// TIA Portal V18 export
DATA_BLOCK "FB_MES_Monitoring_iDB"   // DB10
// stored: InstanceOfName FB_MES_Monitoring, InstanceOfType FB
"FB_MES_Monitoring"
   // VAR_INPUT
   //    Enable : Bool;
   //    Reset : Bool;
   //    HeartbeatTimeout_MES : Time;
   //    HeartbeatTimeout_PLC : Time;
   //    CheckInTimeout : Time;
   //    CheckOutTimeout : Time;
   //    StoveCheckInTimeout : Time;
   // END_VAR
   // VAR_IN_OUT
   //    Diag : "UDT_MES_Monitoring";
   // END_VAR
   // VAR
   //    _hbMesValue : Bool;
   //    _hbPlcValue : Bool;
   //    _errCode : Array[1..8] of DInt;
   //    _errText : Array[1..8] of String[128];
   //    _actErrIdx : Array[1..8] of Int;
   //    _actErrCnt : Int;
   //    _actErrPos : Int;
   //    _errRotateEnable : Bool;
   //    _tErrRotate { S7_SetPoint := 'True'} : TON_TIME;
   //    _hbMesLast : Bool;
   //    _hbPlcLast : Bool;
   //    _tHbMes { S7_SetPoint := 'True'} : TON_TIME;
   //    _tHbPlc { S7_SetPoint := 'True'} : TON_TIME;
   //    _tCi { S7_SetPoint := 'True'} : Array[1..8] of TON_TIME;
   //    _tCo { S7_SetPoint := 'True'} : Array[1..8] of TON_TIME;
   //    _tStove { S7_SetPoint := 'True'} : TON_TIME;
   //    _ciDonePrev : Array[1..8] of Bool;
   //    _coDonePrev : Array[1..8] of Bool;
   //    _ciOkPrev : Array[1..8] of Bool;
   //    _ciNgPrev : Array[1..8] of Bool;
   //    _coOkPrev : Array[1..8] of Bool;
   //    _coNgPrev : Array[1..8] of Bool;
   //    _ciTimeoutLatched : Array[1..8] of Bool;
   //    _coTimeoutLatched : Array[1..8] of Bool;
   //    _spDonePrev : Array[1..8] of Bool;
   //    _spOkPrev : Array[1..8] of Bool;
   //    _spNgPrev : Array[1..8] of Bool;
   //    _lrDonePrev : Array[1..8] of Bool;
   //    _lrOkPrev : Array[1..8] of Bool;
   //    _lrNgPrev : Array[1..8] of Bool;
   //    _stoveOkPrev : Bool;
   //    _stoveTimeoutLatched : Bool;
   //    _i : Int;
   //    _ciReq : Array[1..8] of Bool;
   //    _ciOk : Array[1..8] of Bool;
   //    _ciNg : Array[1..8] of Bool;
   //    _ciDone : Array[1..8] of Bool;
   //    _coReq : Array[1..8] of Bool;
   //    _coOk : Array[1..8] of Bool;
   //    _coNg : Array[1..8] of Bool;
   //    _coDone : Array[1..8] of Bool;
   //    _spOk : Array[1..8] of Bool;
   //    _spNg : Array[1..8] of Bool;
   //    _spDone : Array[1..8] of Bool;
   //    _lrOk : Array[1..8] of Bool;
   //    _lrNg : Array[1..8] of Bool;
   //    _lrDone : Array[1..8] of Bool;
   //    _stoveReq : Bool;
   //    _stoveOk : Bool;
   // END_VAR
BEGIN
END_DATA_BLOCK
